# EPICS substitutions: viocs/substitutions/sd1k.substitutions
file "db/individual.db" {
    pattern { family, pos }
        { "SD1K", "01C4" }
        { "SD1K", "02C4" }
        { "SD1K", "03C4" }
        { "SD1K", "04C4" }
        { "SD1K", "05C4" }
        { "SD1K", "06C4" }
        { "SD1K", "07C4" }
        { "SD1K", "08C4" }
        { "SD1K", "09C4" }
        { "SD1K", "10C4" }
        { "SD1K", "11C4" }
        { "SD1K", "12C4" }
        { "SD1K", "13C4" }
        { "SD1K", "14C4" }
        { "SD1K", "15C4" }
        { "SD1K", "16C4" }
        { "SD1K", "17C4" }
        { "SD1K", "18C4" }
        { "SD1K", "19C4" }
        { "SD1K", "20C4" }
}
